(* IEC 61131-3 sources: CodesysTest/export/Function Blocks, 8 files *)

(* ---- FN_RandomDINT.pou.st ---- *)
(*#-#-#-#-#-#-#-#-#-#---Declaration---#-#-#-#-#-#-#-#-#-#-#-#-#*)

FUNCTION FN_RandomDINT : DINT
VAR_INPUT
	last : DINT;
	low : DINT;
	high : DINT;
END_VAR
VAR
END_VAR
(*#-#-#-#-#-#-#-#-#-#---Implementation---#-#-#-#-#-#-#-#-#-#-#-#-#*)

FN_RandomDINT := TO_DINT(OSCAT_BASIC.RDM(OSCAT_BASIC.FRACT(TO_REAL(last) * OSCAT_BASIC.Globale_Variablen.MATH.PI)) * (TO_REAL(high) - TO_REAL(low) + 1)) + low;

(* ---- FB_GetTime.pou.st ---- *)
(*#-#-#-#-#-#-#-#-#-#---Declaration---#-#-#-#-#-#-#-#-#-#-#-#-#*)

FUNCTION_BLOCK FB_GetTime
VAR_INPUT
END_VAR
VAR_OUTPUT
    currentDateAndTime : DATE_AND_TIME;
END_VAR
VAR
    iState : INT;
    udiUtcTime : UDINT;
    udiUtcTimeLocal : UDINT;
    strTimeDate : SYSTIMEDATE;
    strTimeDateLocal : SYSTIMEDATE;
    dtDateTimeUTC : DATE_AND_TIME;
    timeLeftTime : TIME;
    timeLeftDWORD : DWORD;
    dDateUTC : DATE;
    todTimeOfDayUTC : TOD;

    tSysStartTime : TIME;
    systimeStartNano : SYSTIME;
    udiStartTimeResult : UDINT;
    udiResult : UDINT;

    GetDateAndTime : DTU.GetDateAndTime;
    SetTimeZoneInformation : DTU.SetTimeZoneInformation;

    dtCurrent : DATE_AND_TIME;
    dtConcated : DATE_AND_TIME;
    //eWeekday                 : RTCLK.WEEKDAY;
    uiYear : UINT;
    uiMonth : UINT;
    uiDay : UINT;
    uiHour : UINT;
    uiMinute : UINT;
    uiSecond : UINT;

    dtuError : DTU.ERROR;
END_VAR
(*#-#-#-#-#-#-#-#-#-#---Implementation---#-#-#-#-#-#-#-#-#-#-#-#-#*)

CASE iState OF

    0:
        iState:= 1;

    1:  // retrieves the target date and time, including the timezone information which was set before
        GetDateAndTime( xExecute:= TRUE);
        IF GetDateAndTime.xDone THEN
            dtCurrent:= GetDateAndTime.dtDateAndTime;
            GetDateAndTime(xExecute:= FALSE);
			currentDateAndTime := dtCurrent;
            //timeLeft := TIME_TO_DT(DT_TO_TIME(targetDate) - DT_TO_TIME(dttarget));
            iState:= 2;
        END_IF
        IF GetDateAndTime.xError THEN
            GetDateAndTime(xExecute:= FALSE);
            iState:= 32767;
        END_IF

    2: (*set a spedific date and time --> returns a variable of type DATE_AND_TIME
         DateConcat --> set only date information --> returns a variable of type DATE
         TODConcat  --> set only the time information  --> returns a variable of TOD (Time of day) *)
        IF dtuError = 0 THEN
            iState := 3;
        ELSE
            iState := 32767;
        END_IF

    3:  (*a DATE_AND_TIME variable is splitted in its parts, like year, month, day etc.
            DateSplit --> the same function for a DATE variable
            TODSplit  --> the same function for a TOD variable *)

        IF dtuError = 0 THEN
            iState:= 1;
        ELSE
            iState:= 32767;
        END_IF

    32767: ; //error

END_CASE

(* ---- FB_HMIData.pou.st ---- *)
(*#-#-#-#-#-#-#-#-#-#---Declaration---#-#-#-#-#-#-#-#-#-#-#-#-#*)

{attribute 'FBVisuCreator'}
FUNCTION_BLOCK FB_HMIData
VAR_INPUT
	initiateCycle : BOOL;  // Initiate Cycle Pushbutton
	ackAllFaults : BOOL; // Acknowledge All Faults from HMI
	makeReady : BOOL;
	pressureBarService : ServiceCommands;
	loadPlateService : ServiceCommands;
    stopMachine : BOOL;
	{attribute 'FBVisuCreatorFormatString' := '%s'}
	version : STRING := '0.2A';
	inCycle : BOOL;
	batchEnable : BOOL;
	{attribute 'FBVisuCreatorFormatString' := '%d'}
	batchSetting : UDINT := 10;
	{attribute 'FBVisuCreatorFormatString' := '%d'}
	batchCount : UDINT;
	{attribute 'FBVisuCreatorFormatString' := '%d'}
	headCycleCount : UDINT;
	{attribute 'FBVisuCreatorFormatString' := '%1.2f'}
	pressureBarOpenDelay : REAL;
	{attribute 'FBVisuCreatorFormatString' := '%1.2f'}
	pressureBarCloseDelay : REAL;
	{attribute 'FBVisuCreatorFormatString' := '%1.2f'}
	passthroughSetting : REAL := 8.0;
	{attribute 'FBVisuCreatorFormatString' := '%1.2f'}
	passthroughActual : REAL;
	{attribute 'FBVisuCreatorFormatString' := '%1.2f'}
	lpaDwell : REAL;
	{attribute 'FBVisuCreatorFormatString' := '%1.2f'}
	hpaDwell : REAL;
	{attribute 'FBVisuCreatorFormatString' := '%1.2f'}
	sealBarDwell : REAL := 0.750;
	{attribute 'FBVisuCreatorFormatString' := '%d'}
	sealBarTemperatureSetting : UDINT;
	{attribute 'FBVisuCreatorFormatString' := '%d'}
	sealBarTemperature : UDINT;
	{attribute 'FBVisuCreatorFormatString' := '%1.2f'}
	sealFlattenerBagOpenPositionSetting : REAL;
	{attribute 'FBVisuCreatorFormatString' := '%1.2f'}
	sealFlattenerFlattenedPositionSetting : REAL;
	{attribute 'FBVisuCreatorFormatString' := '%1.2f'}
	sealFlattenerMoveInPositionSetting : REAL;
	{attribute 'FBVisuCreatorFormatString' := '%1.2f'}
	bagSkirtLength : REAL := 1.35;
	{attribute 'FBVisuCreatorFormatString' := '%1.2f'}
	bagLength : REAL := 23.5;
	{attribute 'FBVisuCreatorFormatString' := '%1.2f'}
	bagWidth : REAL := 17.5;
	{attribute 'FBVisuCreatorFormatString' := '%1.2f'}
	bagThickness : REAL := 2.5;
	{attribute 'FBVisuCreatorFormatString' := '%d'}
	bagForwardSpeed : UDINT := 55;
	{attribute 'FBVisuCreatorFormatString' := '%d'}
	bagReverseSpeed : UDINT := 3;
	{attribute 'FBVisuCreatorFormatString' := '%d'}
	printSpeed : UDINT := 6;
	{attribute 'FBVisuCreatorFormatString' := '%1.2f'}
	printLength : REAL := 8.0;
	{attribute 'FBVisuCreatorFormatString' := '%1.2f'}
	printOffset : REAL := 2.0;
	{attribute 'FBVisuCreatorFormatString' := '%d'}
	fillerCountSetting : UDINT;
	{attribute 'FBVisuCreatorFormatString' := '%d'}
	fillerCurrentCount : UDINT;
	{attribute 'FBVisuCreatorFormatString' := '%1.2f'}
	fillerDropTime : REAL;
	{attribute 'FBVisuCreatorFormatString' := '%1.2f'}
	loadPlateDelay : REAL;
	{attribute 'FBVisuCreatorFormatString' := '%1.2f'}
	loadPlateDwell : REAL := 2.5;
	exitConveyorService: ServiceCommands;
	{attribute 'FBVisuCreatorFormatString' := '%1.2f'}
	exitConveyorDwell : REAL := 9.0;
	{attribute 'FBVisuCreatorFormatString' := '%1.2f'}
	lastCycleTime : REAL;
	{attribute 'FBVisuCreatorFormatString' := '%1.2f'}
	bagDropClearanceDwell : REAL := 0.5;
	{attribute 'FBVisuCreatorFormatString' := '%1.2f'}
	averageCycleTime : REAL;
	resetAverageCycleTime : BOOL;
	{attribute 'FBVisuCreatorFormatString' := '%d'}
	bagOpenRetrySetting : UINT := 3;
	{attribute 'FBVisuCreatorFormatString' := '%d'}
	bagOpenRetryCount : UINT;
	{attribute 'FBVisuCreatorFormatString' := '%d'}
	currentJobID : INT;
	separateBeforeSeal : BOOL := TRUE;
	activateDemoMode : BOOL;
	bagOpenAssistEnable : BOOL := TRUE;
	bagOpenSensorEnable : BOOL := TRUE;
	{attribute 'FBVisuCreatorFormatString' := '%1.2f'}
	grabBagDelay : REAL := 0.5;
	{attribute 'FBVisuCreatorFormatString' := '%1.2f'}
	checkForBagOpenDelay : REAL := 1.0;
	{attribute 'FBVisuCreatorFormatString' := '%1.2f'}
	bagClearedFromFingersDelay : REAL := 0.5;
	{attribute 'FBVisuCreatorFormatString' := '%1.2f'}
	vacuumDwell : REAL := 0.5;
	(*Faults*)
	{attribute 'FBVisuCreatorFormatString' := '%s'}
	pressureBarState : STRING;
    stationValveSelection : ARRAY[1..16] OF ValveSelection := 	[ValveSelection.PressureBar,
																ValveSelection.PressureBar,
																ValveSelection.SealBar,
																ValveSelection.HPA_LPA,
																ValveSelection.LoadPlate,
																ValveSelection.BagOpenFingers,
																ValveSelection.PrintHead,
																ValveSelection.Vacuum,
																ValveSelection.SealFlattenersVerticalAxis,
																ValveSelection.LoadShelf,
																6(ValveSelection.Blank)];
    (*Counters*)
    //baggerCycles : FB_MachineCounter(name := 'Bagger Cycle Counter');
	pressureBarCycles : FB_MachineCounter(name := 'Pressure Bar Cycle Counter');
	//passthroughChanges : FB_MachineCounter(name := 'Passthrough Changes Counter');
	//loadPlateCycles : FB_MachineCounter(name := 'Load Plate Cycle Counter');
	//printerCycles : FB_MachineCounter(name := 'Printer Cycle Counter');
	//motorizedSealFlattenerCycles : FB_MachineCounter(name := 'Motorized Seal Flattener Cycles');
	//bagOpenRetryTotal : FB_MachineCounter(name := 'Bag Open Retry Totals');
	(*Info*)
	faultActive : BOOL;
	simulateAllIO : BOOL;

	(*Factoy Config*)
	bofSelection : BagOpenFingersSelection := BagOpenFingersSelection.PneumaticWithBagOpenSensors;
	bofEnable : BOOL := TRUE;
	sealFlattenersSelection : SealFlattenerSelection := SealFlattenerSelection.MotorizedSealFlatteners;
	sealFlattenersEnable : BOOL := TRUE;
	printerSelection : LabelPrinterSelection := LabelPrinterSelection.ZebraPrinter;
	printerEnable : BOOL := TRUE;
	integratedExitConveyorSelection : IntegratedConveyorSelection := IntegratedConveyorSelection.RearExit;
	integratedExitConveyorEnable : BOOL := TRUE;
	packageEjectSelection : PackageEjectionSelection := PackageEjectionSelection.RearRetractingLoadPlate;
	packageEjectEnable : BOOL := TRUE;
END_VAR
VAR_OUTPUT
END_VAR
VAR
END_VAR
(*#-#-#-#-#-#-#-#-#-#---Implementation---#-#-#-#-#-#-#-#-#-#-#-#-#*)

(* ---- FB_LoggableBool.pou.st ---- *)
(*#-#-#-#-#-#-#-#-#-#---Declaration---#-#-#-#-#-#-#-#-#-#-#-#-#*)

FUNCTION_BLOCK FB_LoggableBool EXTENDS FB_BaseObject IMPLEMENTS ILoggable
VAR_INPUT
	in : BOOL;
END_VAR
VAR_OUTPUT
	Q : BOOL;
END_VAR
VAR
END_VAR
(*#-#-#-#-#-#-#-#-#-#---Implementation---#-#-#-#-#-#-#-#-#-#-#-#-#*)

(* ---- FB_MetricConversions.pou.st ---- *)
(*#-#-#-#-#-#-#-#-#-#---Declaration---#-#-#-#-#-#-#-#-#-#-#-#-#*)

FUNCTION_BLOCK e
VAR_INPUT
    bagLengthIn : REAL;
    bagWidthIn : REAL;
    bagSkirtLengthIn : REAL;
    sealBarTempIn : REAL;
    printSpeedIn : UDINT;
    printOffsetIn : REAL;
    printLengthIn : REAL;
    passthroughSettingIn : REAL;
    jawClosePositionSettingIn : REAL;
    barcodeStartPositionIn : REAL;
    barcodeScanningDistanceIn : REAL;
	feedSpeedIn : REAL;
    reverseSpeedIn : REAL;
END_VAR
VAR_OUTPUT
    bagLengthOut : REAL;
    bagWidthOut : REAL;
    bagSkirtLengthOut : REAL;
    sealBarTempOut : REAL;
    printSpeedOut : UDINT;
    printOffsetOut : REAL;
    printLengthOut : REAL;
    passthroughSettingOut : REAL;
    jawClosePositionSettingOut : REAL;
    barcodeStartPositionOut : REAL;
    barcodeScanningDistanceOut : REAL;
   	feedSpeedOut : REAL;
    reverseSpeedOut : REAL;
END_VAR
VAR
    _ConvertMetricToInch: F_TRIG;
    _ConvertInchToMetric: R_TRIG;
END_VAR(*#-#-#-#-#-#-#-#-#-#---Implementation---#-#-#-#-#-#-#-#-#-#-#-#-#*)

//    Function Block: FB_ModbusDWORD
//    Description: Automatically converts inches to mm every time an inch value changes.
//
//    Created by: Steve Olson
//    Created Date: Friday, January 3, 2025

_ConvertInchToMetric(CLK := HMIData.HMIMetric);
_ConvertMetricToInch(CLK := HMIData.HMIMetric);

IF HMIData.HMIMetric THEN
    bagLengthOut := bagLengthIn / 25.4;
    bagWidthOut := bagWidthIn / 25.4;
    bagSkirtLengthOut := bagSkirtLengthIn / 25.4;
    printSpeedOut := LREAL_TO_UDINT(printSpeedIn / 25.4);
    printOffsetOut := printOffsetIn / 25.4;
    printLengthOut := printLengthIn / 25.4;
    passthroughSettingOut := passthroughSettingIn / 25.4;
    jawClosePositionSettingOut := jawClosePositionSettingIn / 25.4;
    barcodeStartPositionOut := barcodeStartPositionIn / 25.4;
    sealBarTempOut := (sealBarTempIn - 32) * 5 / 9; // Fahrenheit to Celsius
    feedSpeedOut := (feedSpeedIn / 25.4);
    reverseSpeedOut := (reverseSpeedIn / 25.4);
ELSE
    bagLengthOut := bagLengthIn;
    bagWidthOut := bagWidthIn;
    bagSkirtLengthOut := bagSkirtLengthIn;
    printSpeedOut := printSpeedIn;
    printOffsetOut := printOffsetIn;
    printLengthOut := printLengthIn;
    passthroughSettingOut := passthroughSettingIn;
    jawClosePositionSettingOut := jawClosePositionSettingIn;
    barcodeStartPositionOut := barcodeStartPositionIn;
    sealBarTempOut := sealBarTempIn;
    feedSpeedOut := feedSpeedIn;
    reverseSpeedOut := reverseSpeedIn;
END_IF

HMIData.HMIMetric; // testing visibility

IF _ConvertInchToMetric.Q THEN
    HMIData.bagLength := bagLengthIn * 25.4;
    HMIData.bagSkirtLength := bagSkirtLengthIn * 25.4;
    HMIData.printOffset := printOffsetIn * 25.4;
    HMIData.printLength := printLengthIn * 25.4;
    HMIData.passthroughSetting := passthroughSettingIn * 25.4;
    HMIData.jawClosePositionSetting := jawClosePositionSettingIn * 25.4;
    HMIData.barcodeStartPosition := barcodeStartPositionIn * 25.4;
	HMIData.printSpeed := REAL_TO_UINT(printSpeedIn * 25.4);
    //sealBarTempOut := (sealBarTempIn - 32) * 5 / 9; // Fahrenheit to Celsius
    HMIData.bagForwardSpeed := REAL_TO_UDINT(feedSpeedIn * 25.4);
    HMIData.bagReverseSpeed := REAL_TO_UDINT(reverseSpeedIn * 25.4);
END_IF

IF _ConvertMetricToInch.Q THEN
    HMIData.bagLength := bagLengthIn / 25.4;
    HMIData.bagSkirtLength := bagSkirtLengthIn / 25.4;
    HMIData.printOffset := printOffsetIn / 25.4;
    HMIData.printLength := printLengthIn / 25.4;
    HMIData.passthroughSetting := passthroughSettingIn / 25.4;
    HMIData.jawClosePositionSetting := jawClosePositionSettingIn / 25.4;
    HMIData.barcodeStartPosition := barcodeStartPositionIn / 25.4;
	HMIData.printSpeed := REAL_TO_UINT(printSpeedIn / 25.4);
    sealBarTempOut := (sealBarTempIn * 9 / 5) + 32; // Celsius to Fahrenheit
    HMIData.bagForwardSpeed := REAL_TO_UDINT(feedSpeedIn / 25.4);
    HMIData.bagReverseSpeed := REAL_TO_UDINT(reverseSpeedIn / 25.4);
END_IF

(* ---- FB_PredictiveMaint.pou.st ---- *)
(*#-#-#-#-#-#-#-#-#-#---Declaration---#-#-#-#-#-#-#-#-#-#-#-#-#*)

FUNCTION_BLOCK FB_PredictiveMaint EXTENDS FB_CycleCounter
VAR_INPUT
	target : UDINT;
	name : STRING;
	units : STRING := 'Machine Cycles';
END_VAR
VAR_OUTPUT

END_VAR
VAR

END_VAR
(*#-#-#-#-#-#-#-#-#-#---Implementation---#-#-#-#-#-#-#-#-#-#-#-#-#*)

SUPER^();

(* ---- FB_SimulatedFeedback.pou.st ---- *)
(*#-#-#-#-#-#-#-#-#-#---Declaration---#-#-#-#-#-#-#-#-#-#-#-#-#*)

FUNCTION_BLOCK FB_SimulatedFeedback EXTENDS FB_BaseObject
VAR_INPUT
	in : BOOL;			// Start of feedback (usually an output)
	simFeedbackFault : BOOL;	// Enable a feedback fault
	faultDelay : DINT;			// Delay for feedback fault
	minDelay : DINT;	//Minimum delay in mS
	maxDelay : DINT;	//Maximum delay in mS
END_VAR
VAR_OUTPUT
	Q : BOOL;
	fault : BOOL;
END_VAR
VAR
	inONS : FB_ONS();
	QONS : FB_ONS();
	_beginTimer : BOOL;
	randomDelay : DINT;
	delayTimer : Standard.TON;
END_VAR
(*#-#-#-#-#-#-#-#-#-#---Implementation---#-#-#-#-#-#-#-#-#-#-#-#-#*)

//	Function Block: FB_SimulatedFeedback
//	Description: Meant to simulate a feedback based off an input with an additional option to simulate a failed feedback signal
//				 Can be used for testing or for creating "feedback" for components that lack a sensor
//
//	Usage: simPbarInFB(in := movePbarInOutput, minDelay := 100, maxDelay := 200);
//
//	Created by: Ben Hess
//	Created Date: 3-2019

inONS(CLK := in);
QONS(CLK := Q);
IF minDelay < 0 THEN
	minDelay := 0;
END_IF
IF inONS.OSR THEN
	_logger.AddLogItem(CONCAT(_prefix,'Started'));
	// Feeback can be set as a range to simulate variations in air pressure, friction etc.
	// Choose a random delay in between min and max
	IF NOT simFeedbackFault THEN
		randomDelay := 	FN_RandomDINT(last := randomDelay,
								low := minDelay,
								high := maxDelay);
		delayTimer.PT := DINT_TO_TIME(randomDelay);
	ELSE
		// Use fault timer if fault sim enabled
		delayTimer.PT := DINT_TO_TIME(faultDelay);
	END_IF
END_IF

IF QONS.OSR AND NOT simFeedbackFault THEN
	_logger.AddLogItem(CONCAT(_prefix,'Done'));
END_IF

delayTimer(IN := in);

IF NOT simFeedbackFault THEN
	Q := delayTimer.Q;
	fault := FALSE;
ELSE
	Q := FALSE;
	fault := delayTimer.Q;
END_IF

(* ---- FB_SimulatedFeedbackPhysicalInput.pou.st ---- *)
(*#-#-#-#-#-#-#-#-#-#---Declaration---#-#-#-#-#-#-#-#-#-#-#-#-#*)

FUNCTION_BLOCK FB_SimulatedFeedbackPhysicalInput EXTENDS FB_SimulatedFeedback
VAR_INPUT
	inputToSimulate : REFERENCE TO FB_PhysicalDigitalInput;
END_VAR
VAR_OUTPUT
END_VAR
VAR
END_VAR
(*#-#-#-#-#-#-#-#-#-#---Implementation---#-#-#-#-#-#-#-#-#-#-#-#-#*)

//	Function Block: FB_SimulatedFeedbackPhysicalInput
//	Description: Meant to simulate a feedback based off an input with an additional option to simulate a failed feedback signal
//				 Using a physical input to simulate
//
//	Usage: simPbarInFB(in := movePbarInOutput, minDelay := 100, maxDelay := 200);
//
//	Created by: Ben Hess
//	Created Date: 5-20-2019

SUPER^();

IF inputToSimulate.simulate = TRUE THEN
	inputToSimulate.simValue := Q;
END_IF
